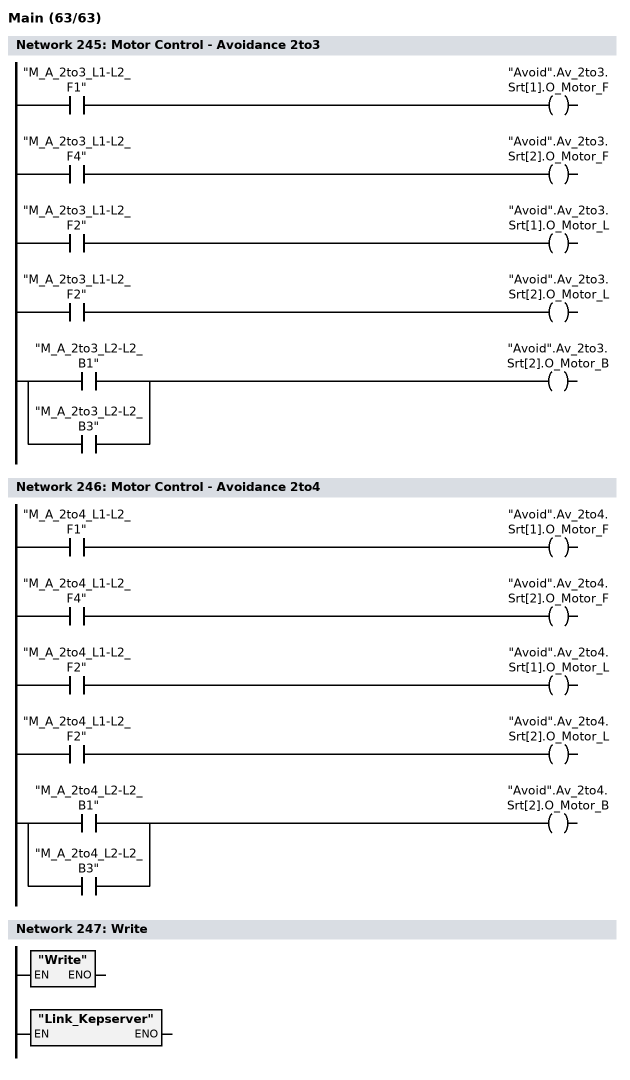
   RUNG wire#powerrail
      Contact( "M_A_2to3_L1-L2_F1" )
      Coil( "Avoid".Av_2to3.Srt[1].O_Motor_F )
   END_RUNG
   RUNG wire#powerrail
      Contact( "M_A_2to3_L1-L2_F4" )
      Coil( "Avoid".Av_2to3.Srt[2].O_Motor_F )
   END_RUNG
   RUNG wire#powerrail
      Contact( "M_A_2to3_L1-L2_F2" )
      Coil( "Avoid".Av_2to3.Srt[1].O_Motor_L )
   END_RUNG
   RUNG wire#powerrail
      Contact( "M_A_2to3_L1-L2_F2" )
      Coil( "Avoid".Av_2to3.Srt[2].O_Motor_L )
   END_RUNG
   RUNG wire#powerrail
      Contact( "M_A_2to3_L2-L2_B1" )
      wire#w1
      Coil( "Avoid".Av_2to3.Srt[2].O_Motor_B )
   END_RUNG
   RUNG wire#powerrail
      Contact( "M_A_2to3_L2-L2_B3" )
   END_RUNG wire#w1
   // the same network as SCL:
   "Avoid".Av_2to3.Srt[1].O_Motor_F := "M_A_2to3_L1-L2_F1";
   "Avoid".Av_2to3.Srt[2].O_Motor_F := "M_A_2to3_L1-L2_F4";
   "Avoid".Av_2to3.Srt[1].O_Motor_L := "M_A_2to3_L1-L2_F2";
   "Avoid".Av_2to3.Srt[2].O_Motor_L := "M_A_2to3_L1-L2_F2";
   "Avoid".Av_2to3.Srt[2].O_Motor_B := "M_A_2to3_L2-L2_B1" OR "M_A_2to3_L2-L2_B3";
END_REGION

REGION Network 246: Motor Control - Avoidance 2to4
   RUNG wire#powerrail
      Contact( "M_A_2to4_L1-L2_F1" )
      Coil( "Avoid".Av_2to4.Srt[1].O_Motor_F )
   END_RUNG
   RUNG wire#powerrail
      Contact( "M_A_2to4_L1-L2_F4" )
      Coil( "Avoid".Av_2to4.Srt[2].O_Motor_F )
   END_RUNG
   RUNG wire#powerrail
      Contact( "M_A_2to4_L1-L2_F2" )
      Coil( "Avoid".Av_2to4.Srt[1].O_Motor_L )
   END_RUNG
   RUNG wire#powerrail
      Contact( "M_A_2to4_L1-L2_F2" )
      Coil( "Avoid".Av_2to4.Srt[2].O_Motor_L )
   END_RUNG
   RUNG wire#powerrail
      Contact( "M_A_2to4_L2-L2_B1" )
      wire#w1
      Coil( "Avoid".Av_2to4.Srt[2].O_Motor_B )
   END_RUNG
   RUNG wire#powerrail
      Contact( "M_A_2to4_L2-L2_B3" )
   END_RUNG wire#w1
   // the same network as SCL:
   "Avoid".Av_2to4.Srt[1].O_Motor_F := "M_A_2to4_L1-L2_F1";
   "Avoid".Av_2to4.Srt[2].O_Motor_F := "M_A_2to4_L1-L2_F4";
   "Avoid".Av_2to4.Srt[1].O_Motor_L := "M_A_2to4_L1-L2_F2";
   "Avoid".Av_2to4.Srt[2].O_Motor_L := "M_A_2to4_L1-L2_F2";
   "Avoid".Av_2to4.Srt[2].O_Motor_B := "M_A_2to4_L2-L2_B1" OR "M_A_2to4_L2-L2_B3";
END_REGION

REGION Network 247: Write
   RUNG wire#powerrail
      "Write"()
   END_RUNG
   RUNG wire#powerrail
      "Link_Kepserver"()
   END_RUNG
   // the same network as SCL:
   "Write"();
   "Link_Kepserver"();
END_REGION
END_ORGANIZATION_BLOCK

(* ===== HMI "HMI_RT_1" =====
system functions are stored by id; their names below are inferred from use
connection "HMI_Connection_1": ETHERNET, SMART_S7_1200_OMS

HMI tags "Default tag table"
   "Boxes_Boxes[1].V_SentFrom" : DInt = PLC Boxes.Boxes[1].V_SentFrom, 1 s
   "Boxes_Boxes[1].V_SectionOn" : DInt = PLC Boxes.Boxes[1].V_SectionOn, 1 s
   "Boxes_Boxes[1].V_ConveyorOn" : DInt = PLC Boxes.Boxes[1].V_ConveyorOn, 1 s
   "Boxes_Boxes[1].V_TypeOn" : Byte = PLC Boxes.Boxes[1].V_TypeOn, 1 s
   "Boxes_Boxes[1].V_Direction" : Byte = PLC Boxes.Boxes[1].V_Direction, 1 s
   "Boxes_Boxes[2].V_SentFrom" : DInt = PLC Boxes.Boxes[2].V_SentFrom, 1 s
   "Boxes_Boxes[2].V_SectionOn" : DInt = PLC Boxes.Boxes[2].V_SectionOn, 1 s
   "Boxes_Boxes[2].V_ConveyorOn" : DInt = PLC Boxes.Boxes[2].V_ConveyorOn, 1 s
   "Boxes_Boxes[2].V_TypeOn" : Byte = PLC Boxes.Boxes[2].V_TypeOn, 1 s
   "Boxes_Boxes[2].V_Direction" : Byte = PLC Boxes.Boxes[2].V_Direction, 1 s
   "Boxes_Boxes[3].V_SentFrom" : DInt = PLC Boxes.Boxes[3].V_SentFrom, 1 s
   "Boxes_Boxes[3].V_SectionOn" : DInt = PLC Boxes.Boxes[3].V_SectionOn, 1 s
   "Boxes_Boxes[3].V_ConveyorOn" : DInt = PLC Boxes.Boxes[3].V_ConveyorOn, 1 s
   "Boxes_Boxes[3].V_TypeOn" : Byte = PLC Boxes.Boxes[3].V_TypeOn, 1 s
   "Boxes_Boxes[3].V_Direction" : Byte = PLC Boxes.Boxes[3].V_Direction, 1 s
   "Boxes_Boxes[4].V_SentFrom" : DInt = PLC Boxes.Boxes[4].V_SentFrom, 1 s
   "Boxes_Boxes[4].V_SectionOn" : DInt = PLC Boxes.Boxes[4].V_SectionOn, 1 s
   "Boxes_Boxes[4].V_ConveyorOn" : DInt = PLC Boxes.Boxes[4].V_ConveyorOn, 1 s
   "Boxes_Boxes[4].V_TypeOn" : Byte = PLC Boxes.Boxes[4].V_TypeOn, 1 s
   "Boxes_Boxes[4].V_Direction" : Byte = PLC Boxes.Boxes[4].V_Direction, 1 s
   "Boxes_Boxes[5].V_SentFrom" : DInt = PLC Boxes.Boxes[5].V_SentFrom, 1 s
   "Boxes_Boxes[5].V_SectionOn" : DInt = PLC Boxes.Boxes[5].V_SectionOn, 1 s
   "Boxes_Boxes[5].V_ConveyorOn" : DInt = PLC Boxes.Boxes[5].V_ConveyorOn, 1 s
   "Boxes_Boxes[5].V_TypeOn" : Byte = PLC Boxes.Boxes[5].V_TypeOn, 1 s
   "Boxes_Boxes[5].V_Direction" : Byte = PLC Boxes.Boxes[5].V_Direction, 1 s
   "B_Pharmacy_ChooseRoom" : Bool = PLC B_Pharmacy_ChooseRoom AT %M0.1, 1 s
   "B_Pharmacy_Go" : Bool = PLC B_Pharmacy_Go AT %M0.2, 1 s
   "B_Pharmacy_Room1" : Int = PLC B_Pharmacy_Room1 AT %MW2, 1 s
   "B_Pharmacy_Room2" : Int = PLC B_Pharmacy_Room2 AT %MW4, 1 s
   "B_Pharmacy_Room3" : Int = PLC B_Pharmacy_Room3 AT %MW6, 1 s
   "B_Pharmacy_Start" : Bool = PLC B_Pharmacy_Start AT %M0.0, 1 s
   "B_R1_Continue" : Bool = PLC B_R1_Continue AT %M20.2, 1 s
   "B_R1_Return" : Bool = PLC B_R1_Return AT %M20.3, 1 s
   "B_R2_Continue" : Bool = PLC B_R2_Continue AT %M20.4, 1 s
   "B_R2_Return" : Bool = PLC B_R2_Return AT %M20.5, 1 s
   "M_Pharmacy_Start" : Bool = PLC M_Pharmacy_Start AT %M0.4, 1 s
   "M_R1_Start" : Bool = PLC M_R1_Start AT %M17.5, 1 s
   "M_R2_Start" : Bool = PLC M_R2_Start AT %M18.3, 1 s
   "Boxes_Boxes{1}_V_Completed" : Array [0..2] of DInt = PLC Boxes.Boxes[1].V_Completed AT %DB1.DBX0.0, 1 s
   "Boxes_Boxes{1}_V_NumOfComp" : DInt = PLC Boxes.Boxes[1].V_NumOfComp AT %DB1.DBX0.0, 1 s
   "Boxes_Boxes{2}_V_Completed" : Array [0..2] of DInt = PLC Boxes.Boxes[2].V_Completed AT %DB1.DBD0, 1 s
   "Boxes_Boxes{2}_V_NumOfComp" : DInt = PLC Boxes.Boxes[2].V_NumOfComp AT %DB1.DBD0, 1 s
   "Boxes_Boxes{3}_V_Completed" : Array [0..2] of DInt = PLC Boxes.Boxes[3].V_Completed AT %DB1.DBD0, 1 s
   "Boxes_Boxes{3}_V_NumOfComp" : DInt = PLC Boxes.Boxes[3].V_NumOfComp AT %DB1.DBD0, 1 s
   "Boxes_Boxes{4}_V_Completed" : Array [0..2] of DInt = PLC Boxes.Boxes[4].V_Completed AT %DB1.DBD0, 1 s
   "Boxes_Boxes{4}_V_NumOfComp" : DInt = PLC Boxes.Boxes[4].V_NumOfComp AT %DB1.DBD0, 1 s
   "Boxes_Boxes{5}_V_Completed" : Array [0..2] of DInt = PLC Boxes.Boxes[5].V_Completed AT %DB1.DBD0, 1 s
   "Boxes_Boxes{5}_V_NumOfComp" : DInt = PLC Boxes.Boxes[5].V_NumOfComp AT %DB1.DBD0, 1 s
   "R1_has_box" : Bool = PLC R1_has_box AT %M39.0, 1 s
   "R2_has_box" : Bool = PLC R2_has_box AT %M39.1, 1 s

screen "Home" 1280x800, template "Template_1"
   TextField "Text field_1" at 542,78 size 196x79; Text 'HOME'
   Button "Button_1" at 223,240 size 834x75; TextOff 'Pharmacy'
      on Click: ActivateScreen("SIm Pharmacy", 0)
      Appearance <- "M_Pharmacy_Start"
   Button "Button_2" at 223,367 size 834x75; TextOff 'Paediatrics'
      on Click: ActivateScreen("Sim Paediatrics", 0)
      Appearance <- "M_R1_Start"
   Button "Button_3" at 223,493 size 834x75; TextOff 'ICU'
      on Click: ActivateScreen("Sim ICU", 0)
      Appearance <- "M_R2_Start"
   Button "Button_4" at 223,622 size 834x75; TextOff 'Boxes'
      on Click: ActivateScreen("Box Info", 0)
   Button "Button_5" at 1059,367 size 99x75; TextOff 'GET'
      on Click: ResetBit("R1_has_box")
      Appearance <- "R1_has_box"
   Button "Button_6" at 1060,493 size 98x75; TextOff 'GET'
      on Click: ResetBit("R2_has_box")
      Appearance <- "R2_has_box"

screen "Box Info" 1280x800, template "Template_1"
   TextField "Text field_1" at 536,25 size 301x45; Text 'Box Information'
   TextField "Text field_2" at 212,208 size 56x25; Text 'Box 1'
   TextField "Text field_3" at 212,297 size 56x25; Text 'Box 2'
   TextField "Text field_4" at 212,388 size 56x25; Text 'Box 3'
   TextField "Text field_5" at 212,479 size 56x25; Text 'Box 4'
   TextField "Text field_6" at 212,570 size 56x25; Text 'Box 5'
   TextField "Text field_7" at 343,113 size 55x25; Text 'Dest 1'
   TextField "Text field_8" at 449,113 size 55x25; Text 'Dest 2'
   TextField "Text field_9" at 556,113 size 55x25; Text 'Dest 3'
   TextField "Text field_10" at 662,113 size 62x25; Text 'SectOn'
   TextField "Text field_11" at 1016,113 size 67x25; Text 'TypeOn'
   TextField "Text field_12" at 778,113 size 57x25; Text 'CnvOn'
   TextField "Text field_13" at 886,113 size 76x25; Text 'Direction'
   IOField "I/O field_4" at 343,451 size 57x62; FormatPattern 9
      ProcessValue <- "[0]"
      Appearance <- "Boxes_Boxes{4}_V_NumOfComp"
   IOField "I/O field_9" at 449,451 size 57x62; FormatPattern 9
      ProcessValue <- "[1]"
      Appearance <- "Boxes_Boxes{4}_V_NumOfComp"
   IOField "I/O field_14" at 556,451 size 57x62; FormatPattern 9
      ProcessValue <- "[2]"
      Appearance <- "Boxes_Boxes{4}_V_NumOfComp"
   IOField "I/O field_16" at 662,181 size 57x62; FormatPattern 9
      ProcessValue <- "Boxes_Boxes[1].V_SectionOn"
   IOField "I/O field_17" at 662,270 size 57x62; FormatPattern 9
      ProcessValue <- "Boxes_Boxes[2].V_SectionOn"
   IOField "I/O field_18" at 662,361 size 57x62; FormatPattern 9
      ProcessValue <- "Boxes_Boxes[3].V_SectionOn"
   IOField "I/O field_19" at 662,451 size 57x62; FormatPattern 9
      ProcessValue <- "Boxes_Boxes[4].V_SectionOn"
   IOField "I/O field_20" at 662,542 size 57x62; FormatPattern 9
      ProcessValue <- "Boxes_Boxes[5].V_SectionOn"
   TextField "Text field_14" at 1017,210 size 56x25; Text 'Avoid'
      Visibility <- "Boxes_Boxes[1].V_TypeOn"
   TextField "Text field_15" at 995,210 size 94x25; Text 'Up/Down'
      Visibility <- "Boxes_Boxes[1].V_TypeOn"
   TextField "Text field_16" at 1003,210 size 79x25; Text 'Straight'
      Visibility <- "Boxes_Boxes[1].V_TypeOn"
   TextField "Text field_17" at 1017,299 size 56x25; Text 'Avoid'
      Visibility <- "Boxes_Boxes[2].V_TypeOn"
   TextField "Text field_18" at 995,299 size 94x25; Text 'Up/Down'
      Visibility <- "Boxes_Boxes[2].V_TypeOn"
   TextField "Text field_19" at 1003,299 size 79x25; Text 'Straight'
      Visibility <- "Boxes_Boxes[2].V_TypeOn"
   TextField "Text field_20" at 1017,390 size 56x25; Text 'Avoid'
      Visibility <- "Boxes_Boxes[3].V_TypeOn"
   TextField "Text field_21" at 995,390 size 94x25; Text 'Up/Down'
      Visibility <- "Boxes_Boxes[3].V_TypeOn"
   TextField "Text field_22" at 1003,390 size 79x25; Text 'Straight'
      Visibility <- "Boxes_Boxes[3].V_TypeOn"
   TextField "Text field_23" at 1017,481 size 56x25; Text 'Avoid'
      Visibility <- "Boxes_Boxes[4].V_TypeOn"
   TextField "Text field_24" at 995,481 size 94x25; Text 'Up/Down'
      Visibility <- "Boxes_Boxes[4].V_TypeOn"
   TextField "Text field_25" at 1003,481 size 79x25; Text 'Straight'
      Visibility <- "Boxes_Boxes[4].V_TypeOn"
   TextField "Text field_26" at 1017,571 size 56x25; Text 'Avoid'
      Visibility <- "Boxes_Boxes[5].V_TypeOn"
   TextField "Text field_27" at 995,571 size 94x25; Text 'Up/Down'
      Visibility <- "Boxes_Boxes[5].V_TypeOn"
   TextField "Text field_28" at 1003,571 size 79x25; Text 'Straight'
      Visibility <- "Boxes_Boxes[5].V_TypeOn"
   IOField "I/O field_21" at 778,181 size 57x62; FormatPattern 9
      ProcessValue <- "Boxes_Boxes[1].V_ConveyorOn"
   IOField "I/O field_22" at 778,270 size 57x62; FormatPattern 9
      ProcessValue <- "Boxes_Boxes[2].V_ConveyorOn"
   IOField "I/O field_23" at 778,361 size 57x62; FormatPattern 9
      ProcessValue <- "Boxes_Boxes[3].V_ConveyorOn"
   IOField "I/O field_24" at 778,451 size 57x62; FormatPattern 9
      ProcessValue <- "Boxes_Boxes[4].V_ConveyorOn"
   IOField "I/O field_25" at 778,542 size 57x62; FormatPattern 9
      ProcessValue <- "Boxes_Boxes[5].V_ConveyorOn"
   IOField "I/O field_26" at 886,181 size 57x62; FormatPattern 9
      ProcessValue <- "Boxes_Boxes[1].V_Direction"
   IOField "I/O field_27" at 886,270 size 57x62; FormatPattern 9
      ProcessValue <- "Boxes_Boxes[2].V_Direction"
   IOField "I/O field_28" at 886,361 size 57x62; FormatPattern 9
      ProcessValue <- "Boxes_Boxes[3].V_Direction"
   IOField "I/O field_29" at 886,451 size 57x62; FormatPattern 9
      ProcessValue <- "Boxes_Boxes[4].V_Direction"
   IOField "I/O field_30" at 886,542 size 57x62; FormatPattern 9
      ProcessValue <- "Boxes_Boxes[5].V_Direction"
   TextField "Text field_29" at 1027,210 size 41x25; Text 'N/A'
      Visibility <- "Boxes_Boxes[1].V_TypeOn"
   TextField "Text field_30" at 1027,299 size 41x25; Text 'N/A'
      Visibility <- "Boxes_Boxes[2].V_TypeOn"
   TextField "Text field_31" at 1027,390 size 41x25; Text 'N/A'
      Visibility <- "Boxes_Boxes[3].V_TypeOn"
   TextField "Text field_32" at 1027,481 size 41x25; Text 'N/A'
      Visibility <- "Boxes_Boxes[4].V_TypeOn"
   TextField "Text field_33" at 1027,571 size 41x25; Text 'N/A'
      Visibility <- "Boxes_Boxes[5].V_TypeOn"
   Button "Button_1" at 590,693 size 156x52; TextOff 'Home'
      on Click: ActivateScreen("Home", 0)
   IOField "I/O field_5" at 343,542 size 57x62; FormatPattern 9
      Appearance <- "Boxes_Boxes{5}_V_NumOfComp"
      ProcessValue <- "[0]"
   IOField "I/O field_10" at 449,542 size 57x62; FormatPattern 9
      Appearance <- "Boxes_Boxes{5}_V_NumOfComp"
      ProcessValue <- "[1]"
   IOField "I/O field_15" at 556,542 size 57x62; FormatPattern 9
      Appearance <- "Boxes_Boxes{5}_V_NumOfComp"
      ProcessValue <- "[2]"
   IOField "I/O field_3" at 343,361 size 57x62; FormatPattern 9
      Appearance <- "Boxes_Boxes{3}_V_NumOfComp"
      ProcessValue <- "[0]"
   IOField "I/O field_8" at 449,361 size 57x62; FormatPattern 9
      Appearance <- "Boxes_Boxes{3}_V_NumOfComp"
      ProcessValue <- "[1]"
   IOField "I/O field_13" at 556,361 size 57x62; FormatPattern 9
      Appearance <- "Boxes_Boxes{3}_V_NumOfComp"
      ProcessValue <- "[2]"
   IOField "I/O field_2" at 343,270 size 57x62; FormatPattern 9
      Appearance <- "Boxes_Boxes{2}_V_NumOfComp"
      ProcessValue <- "[0]"
   IOField "I/O field_7" at 449,270 size 57x62; FormatPattern 9
      Appearance <- "Boxes_Boxes{2}_V_NumOfComp"
      ProcessValue <- "[1]"
   IOField "I/O field_12" at 556,270 size 57x62; FormatPattern 9
      Appearance <- "Boxes_Boxes{2}_V_NumOfComp"
      ProcessValue <- "[2]"
   IOField "I/O field_1" at 343,181 size 57x62; FormatPattern 9
      Appearance <- "Boxes_Boxes{1}_V_NumOfComp"
      ProcessValue <- "[0]"
   IOField "I/O field_6" at 449,181 size 57x62; FormatPattern 9
      Appearance <- "Boxes_Boxes{1}_V_NumOfComp"
      ProcessValue <- "[1]"
   IOField "I/O field_11" at 556,181 size 57x62; FormatPattern 9
      Appearance <- "Boxes_Boxes{1}_V_NumOfComp"
      ProcessValue <- "[2]"

screen "SIm Pharmacy" 1280x800, template "Template_1"
   TextField "Text field_1" at 297,25 size 686x79; Text 'Pharmacy Simulation'
   Button "Button_1" at 564,681 size 153x51; TextOff 'Home'
      on Click: ActivateScreen("Home", 0)
   Button "Button_2" at 483,265 size 315x67; TextOff 'Choose Room'
      on Press: SetBit("B_Pharmacy_Start")
      on Release: ResetBit("B_Pharmacy_Start"); ActivateScreen("Choose Room", 0)
      Visibility <- "M_Pharmacy_Start"

screen "Sim ICU" 1280x800, template "Template_1"
   TextField "Text field_1" at 396,25 size 488x79; Text 'ICU Simulation'
   Button "Button_1" at 566,666 size 150x50; TextOff 'Home'
      on Click: ActivateScreen("Home", 0)
   Rectangle "Rectangle_1" at 276,170 size 729x454
      Visibility <- "M_R2_Start"
   Button "Button_2" at 455,282 size 371x87; TextOff 'Continue'
      on Release: ResetBit("B_R2_Continue")
      on Press: SetBit("B_R2_Continue")
      Visibility <- "M_R2_Start"
   Button "Button_3" at 455,419 size 371x87; TextOff 'Return'
      on Release: ResetBit("B_R2_Return")
      on Press: SetBit("B_R2_Return")
      Visibility <- "M_R2_Start"

screen "Sim Paediatrics" 1280x800, template "Template_1"
   Button "Button_1" at 566,667 size 150x50; TextOff 'Home'
      on Click: ActivateScreen("Home", 0)
   TextField "Text field_1" at 295,25 size 690x79; Text 'Paediatric Simulation'
   Rectangle "Rectangle_1" at 276,170 size 729x455
      Visibility <- "M_R1_Start"
   Button "Button_2" at 455,282 size 371x87; TextOff 'Continue'
      on Press: SetBit("B_R1_Continue")
      on Release: ResetBit("B_R1_Continue")
      Visibility <- "M_R1_Start"
   Button "Button_3" at 455,419 size 371x87; TextOff 'Return'
      on Release: ResetBit("B_R1_Return")
      on Press: SetBit("B_R1_Return")
      Visibility <- "M_R1_Start"

screen "Choose Room" 1280x800, template "Template_1"
   TextField "Text field_1" at 407,159 size 466x60; Text 'Choose destination'
   Button "Button_1" at 475,567 size 330x124; TextOff 'GO'
      Visibility <- "B_Pharmacy_Room1"
      on Press: SetBit("B_Pharmacy_Go")
      on Release: ResetBit("B_Pharmacy_Go"); ActivateScreen("SIm Pharmacy", 0)
   IOField "I/O field_1" at 738,352 size 111x122; FormatPattern 9
      ProcessValue <- "B_Pharmacy_Room2"
   IOField "I/O field_2" at 432,352 size 111x122; FormatPattern 9
      ProcessValue <- "B_Pharmacy_Room1"
*)